Universal Robots PolyScope program: skinkekutter2.urp

Program skinkekutter2 (installation=skinkekutter2 directory=/programs createdIn=0.0.0 lastSavedIn=5.13.0 robotSerialNumber=20185300015)
Calibrated DH parameters: a=[-0.000086, -0.242565, -0.211836, 0.000046, -0.000137, 0]; d=[0.151986, 5.97615, 11.782146, -17.627443, 0.08527, 0.092315]; alpha=[1.571049, 0.003818, 0.001446, 1.57052, -1.5709, 0]; deltaTheta=[0, 0.093783, 0.026843, -0.120628, 0.00001, 0]
Robot Program (runOnlyOnce=true) Move(motionType=MoveL speed=0.1 acceleration=0.1 useActiveTCP=true positionType=CartesianPose, feature=feature, children(Waypoint(type=Fixed name=served, position(JointAngles=[-1.240999, -0.588828, 0.646334, -1.499566, 1.535617, -1.598437], TCPOffset=[0.05, 0, 0, 0, 0, 0]), BaseToFeature=[0, 0, 0, 0, 0, 0])))
